FUNCTION_BLOCK Mc2MotionHomeTask_SetZeroHere EXTENDS Mc2MotionTask
VAR
	MCSetPosition : Tc2_MC2.MC_SetPosition;
END_VAR

{attribute 'monitoring' := 'call'}
PROPERTY Busy : BOOL
GET
Busy := MCSetPosition.Busy;
END_GET
END_PROPERTY

METHOD CyclicLogic
MCSetPosition(Axis := _Axis.Axis);
MCSetPosition.Execute := FALSE;
END_METHOD

{attribute 'monitoring' := 'call'}
PROPERTY Error : BOOL
GET
Error := MCSetPosition.Error;
END_GET
END_PROPERTY

{attribute 'monitoring' := 'call'}
PROPERTY ErrorId : UDINT
GET
ErrorId := MCSetPosition.ErrorID;
END_GET
END_PROPERTY

METHOD Execute : BOOL
IF Axis.Busy OR Axis.Error THEN
	RETURN;
END_IF

MCSetPosition.Execute := TRUE;
Execute				  := TRUE;
END_METHOD

END_FUNCTION_BLOCK

(* stored: Version 1.1.0.1, ProductVersion 3.1.4026.20
   POU Mc2MotionHomeTask_SetZeroHere: Id {a597f766-7dac-4f85-8368-29d7aa566d60}, SpecialFunc None
   Property Busy: Id {70f336e5-0727-4ab1-ba2e-a0f7358fa81c}
   Get Get: Id {d4b500af-245f-4a36-a462-e6b3da481253}
   Method CyclicLogic: Id {0f448220-2036-4a5f-9da7-7e5e7dcf8fd5}
   Property Error: Id {00d65186-6746-443d-8adb-2db181526186}
   Get Get: Id {062f9d6e-bb0f-431e-bcf9-1275212a589d}
   Property ErrorId: Id {969f7443-1338-4a22-83ca-8ea503e40fe3}
   Get Get: Id {c16a34a5-9452-42dc-8584-66302272f9e2}
   Method Execute: Id {7733f637-ca5c-4c3e-a9a3-f72cb47e5f44} *)
